// TIA Portal project "Grundkurs Aufgabe 9 NEU" (V15.1)
// Vorlageprojekt für das Buch mit Zielsystem S7-1200

(* hardware
DEVICE "S7-1200-Station_1"  S7-1200 Station
   slot 0: "Baugruppenträger_0"  Rack  V1.0
   slot 1: "SPS"  CPU 1212C AC/DC/Rly  6ES7 212-1BE40-0XB0  V4.2
*)

// ===== PLC "SPS"  CPU 1212C AC/DC/Rly =====

VAR_GLOBAL   // PLC tag table "Eingänge und Ausgänge"
   "Lichttaster_Rutsche" AT %E0.0 : Bool;   // Lichttaster auf Förderband bei Rutsche (Schließer)
   "Lichttaster_Stanze" AT %E0.1 : Bool;   // Lichttaster auf Förderband bei Stanze (Schließer)
   "Lichttaster_Ende" AT %E0.2 : Bool;   // Lichttaster auf Förderband am Ende bei Kiste (Schließer)
   "Sensor_Stanze_unten" AT %E0.3 : Bool;   // Stanze hat untere Endlage erreicht (Schließer)
   "Sensor_Zentrierung_zugestellt" AT %E0.4 : Bool;   // Zentrierung wurde zugestellt -> Bauteil ist ausgerichtet (Schließer)
   "Motor_Foerderband_vor" AT %A0.0 : Bool;   // Förderband vorwärts in Richtung Stanze
   "Motor_Foerderband_rueck" AT %A0.1 : Bool;   // Förderband rückwärts in Richtung Kiste
   "Stanze_senken" AT %A0.2 : Bool;   // Stanze nach unten fahren
   "Zentrierung_zustellen" AT %A0.3 : Bool;   // Zentrierung zustellen und Bauteil ausrichten für Stanzvorgang
END_VAR

VAR_GLOBAL   // PLC tag table "Merker"
   "Foerderband_vor" AT %M1.0 : Bool;   // Förderband nach vorne fahren bis Stanze
   "Bauteil_zentrieren" AT %M1.1 : Bool;   // Bauteil zentrieren für Stanzvorgang
   "Stanze_nach_unten" AT %M1.2 : Bool;   // Stanze nach unten fahren
   "Foerderband_rueck" AT %M1.3 : Bool;   // Förderband rückwärts fahren bis Kiste
   "Hilfsmerker_FN1" AT %M100.0 : Bool;   // Hilfsmerker negative Flanke
   "Hilfsmerker_FN2" AT %M100.1 : Bool;   // Hilfsmerker negative Flanke
   "Hilfsmerker_FN3" AT %M100.2 : Bool;   // Hilfsmerker negative Flanke
   "Hilfsmerker_FN4" AT %M100.3 : Bool;   // Hilfsmerker negative Flanke
END_VAR

// folder: System blocks/Program resources

DATA_BLOCK "Einschaltverz_Stanze_rueck"   // DB1
{ S7_Optimized_Access := 'TRUE' }
AUTHOR : Simatic
FAMILY : IEC
NAME : IEC_TMR
VERSION : 1.0
// stored: InstanceOfName IEC_TIMER
"IEC_TIMER"
BEGIN
END_DATA_BLOCK

// folder: (top level)

FUNCTION "Kopplung_FactoryIO_mit_PLCSIM" : Void   // FC9000, SCL
{ S7_Optimized_Access := 'TRUE' }
VERSION : 0.1
   VAR_TEMP
      rdTimeReturn : Int;
      outputTime : DTL;
      SyncVal : Byte;
      forVal : Int;
      forVal_2 : Int;
      Value : Byte;
   END_VAR
   VAR CONSTANT
      CompVal : Byte := 16#34;
      Value_01 : Byte := 16#11;
      Value_01_DW : DWord := 16#A165_D992;
      Value_02_DW : DWord := 16#58BE_4401;
   END_VAR
BEGIN

   #Value:=PEEK(area := 16#82,
        dbNumber := 0,
        byteOffset := 511);
   #Value := #Value + 1;

   POKE(area := 16#82,
        dbNumber := 0,
        byteOffset := 511,
        value := #Value);

   POKE(area:=16#81,
        dbNumber:=0,
        byteOffset:=1016,
        value:=#Value_01_DW);
   POKE(area := 16#81,
        dbNumber := 0,
        byteOffset := 1020,
        value := #Value_02_DW);

   POKE(area := 16#81,
        dbNumber := 0,
        byteOffset := 511,
        value := B#16#00);

   FOR #forVal := 0 TO 120 DO
       FOR #forVal_2:=0 TO 10 DO
           #rdTimeReturn:=RD_SYS_T(#outputTime);
           #rdTimeReturn := WR_SYS_T(#outputTime);
           #rdTimeReturn := RD_SYS_T(#outputTime);
           #rdTimeReturn := WR_SYS_T(#outputTime);
       END_FOR;
       #SyncVal:= PEEK(area := 16#81,
                      dbNumber := 0,
                      byteOffset := 511);
       IF #SyncVal = #CompVal THEN
          GOTO M_1;
       END_IF;
   END_FOR;
   RETURN;

   M_1:
   POKE(area := 16#81,
        dbNumber := 0,
        byteOffset := 511,
        value := B#16#0);
END_FUNCTION

ORGANIZATION_BLOCK "Main"   // OB1, FBD, ProgramCycle
TITLE = "Main Program Sweep (Cycle)"
{ S7_Optimized_Access := 'TRUE' }
VERSION : 0.1
   VAR_INPUT
      Initial_Call : Bool;   // Initial call of this OB
      Remanence : Bool;   // =True, if remanent data are available
   END_VAR
   VAR_TEMP   // added for the SCL form of the ladder/FBD networks
      _w1 : Bool;
      _w2 : Bool;
   END_VAR
BEGIN

REGION Network 1: Konnektierungsbaustein für PLC-Lab / Bausteinaufruf FC9000 (Für Aufgabe nicht relevant)
   // Im Netzwerk 1 wird der Konnektierungsbaustein für PLC-Lab aufgerufen.
   // Dieser Aufruf darf nicht entfernt werden!
   // Der Baustein FC9000 organisiert den Datentransfer zwischen PLCSIM und FactoryIO.
   // Der Baustein kann als Beispielprojekt von der FactoryIO-Homepage heruntergeladen werden.
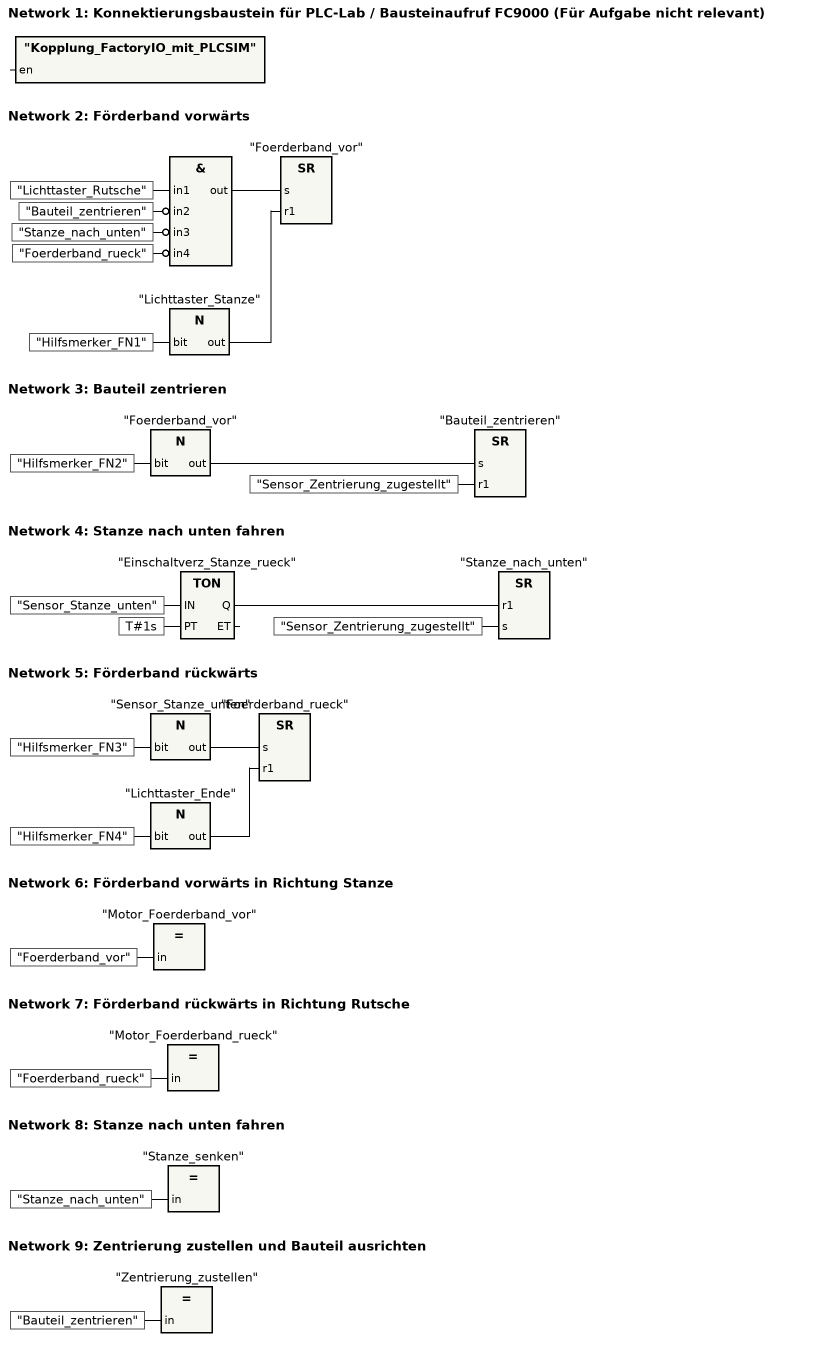
   "Kopplung_FactoryIO_mit_PLCSIM"();
END_REGION

REGION Network 2: Förderband vorwärts
   #_w1 := NOT "Lichttaster_Stanze" AND "Hilfsmerker_FN1";   // falling edge of "Lichttaster_Stanze"
   "Hilfsmerker_FN1" := "Lichttaster_Stanze";
   IF "Lichttaster_Rutsche" AND NOT "Bauteil_zentrieren" AND NOT "Stanze_nach_unten" AND NOT "Foerderband_rueck" THEN
       "Foerderband_vor" := TRUE;   // SR flip-flop
   END_IF;
   IF #_w1 THEN "Foerderband_vor" := FALSE; END_IF;
END_REGION

REGION Network 3: Bauteil zentrieren
   #_w1 := NOT "Foerderband_vor" AND "Hilfsmerker_FN2";   // falling edge of "Foerderband_vor"
   "Hilfsmerker_FN2" := "Foerderband_vor";
   IF #_w1 THEN
       "Bauteil_zentrieren" := TRUE;   // SR flip-flop
   END_IF;
   IF "Sensor_Zentrierung_zugestellt" THEN "Bauteil_zentrieren" := FALSE; END_IF;
END_REGION

REGION Network 4: Stanze nach unten fahren
   "Einschaltverz_Stanze_rueck".TON(IN := "Sensor_Stanze_unten", PT := T#1s);
   IF "Sensor_Zentrierung_zugestellt" THEN
       "Stanze_nach_unten" := TRUE;   // SR flip-flop
   END_IF;
   IF "Einschaltverz_Stanze_rueck".Q THEN "Stanze_nach_unten" := FALSE; END_IF;
END_REGION

REGION Network 5: Förderband rückwärts
   #_w1 := NOT "Sensor_Stanze_unten" AND "Hilfsmerker_FN3";   // falling edge of "Sensor_Stanze_unten"
   "Hilfsmerker_FN3" := "Sensor_Stanze_unten";
   #_w2 := NOT "Lichttaster_Ende" AND "Hilfsmerker_FN4";   // falling edge of "Lichttaster_Ende"
   "Hilfsmerker_FN4" := "Lichttaster_Ende";
   IF #_w1 THEN
       "Foerderband_rueck" := TRUE;   // SR flip-flop
   END_IF;
   IF #_w2 THEN "Foerderband_rueck" := FALSE; END_IF;
END_REGION

REGION Network 6: Förderband vorwärts in Richtung Stanze
   "Motor_Foerderband_vor" := "Foerderband_vor";
END_REGION

REGION Network 7: Förderband rückwärts in Richtung Rutsche
   "Motor_Foerderband_rueck" := "Foerderband_rueck";
END_REGION

REGION Network 8: Stanze nach unten fahren
   "Stanze_senken" := "Stanze_nach_unten";
END_REGION

REGION Network 9: Zentrierung zustellen und Bauteil ausrichten
   "Zentrierung_zustellen" := "Bauteil_zentrieren";
END_REGION
END_ORGANIZATION_BLOCK